FUNCTION_BLOCK SL_Dispense (* Dispense: Requires TRUE; waits Volume / FlowRate s; Invariant TRUE *)
  (* Standard: 61499-2 *)
  (* Version 0.1, 2026-09-28, Project contributors, AAU Smart Production Lab *)
  PACKAGE filling;
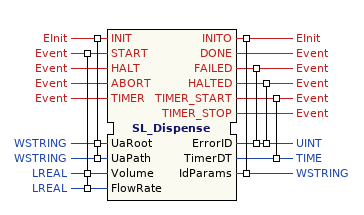
  EVENT_INPUT
    INIT : EInit WITH UaRoot, UaPath;
    START WITH Volume, FlowRate;
    HALT;
    ABORT;
    TIMER;
  END_EVENT
  EVENT_OUTPUT
    INITO : EInit WITH IdParams;
    DONE;
    FAILED WITH ErrorID;
    HALTED WITH ErrorID;
    TIMER_START WITH TimerDT;
    TIMER_STOP;
  END_EVENT
  VAR_INPUT
    UaRoot : WSTRING;
    UaPath : WSTRING;
    Volume : LREAL;
    FlowRate : LREAL;
  END_VAR
  VAR_OUTPUT
    ErrorID : UINT;
    TimerDT : TIME;
    IdParams : WSTRING;
  END_VAR
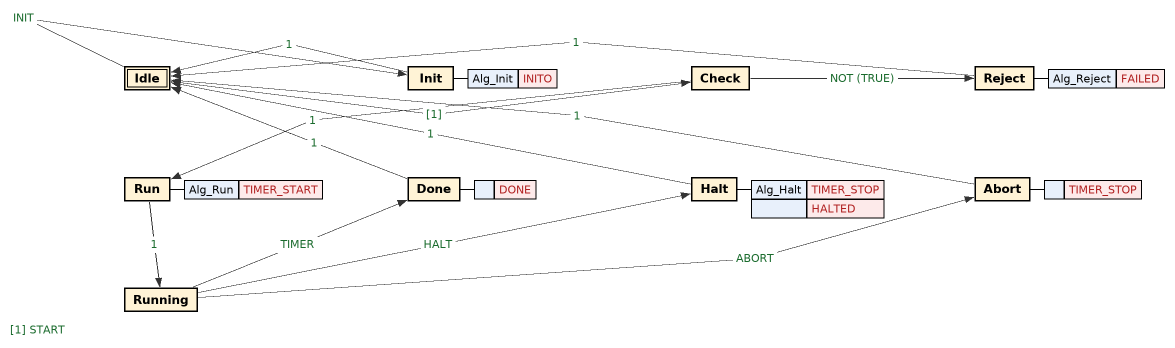
  EC_STATES
    Idle;
    Init : Alg_Init -> INITO;
    Check;
    Reject : Alg_Reject -> FAILED;
    Run : Alg_Run -> TIMER_START;
    Done : -> DONE;
    Halt : Alg_Halt -> TIMER_STOP, -> HALTED;
    Abort : -> TIMER_STOP;
    Running;
  END_STATES
  EC_TRANSITIONS
    Idle TO Init := INIT;
    Init TO Idle := 1;
    Idle TO Check := START;
    Check TO Reject := NOT (TRUE);
    Running TO Done := TIMER;
    Done TO Idle := 1;
    Halt TO Idle := 1;
    Abort TO Idle := 1;
    Check TO Run := 1;
    Run TO Running := 1;
    Running TO Halt := HALT;
    Running TO Abort := ABORT;
    Reject TO Idle := 1;
  END_TRANSITIONS
  ALGORITHM Alg_Init IN ST:
IdParams := CONCAT(CONCAT(CONCAT(CONCAT(CONCAT("opc_ua[WRITE;", CONCAT(UaRoot, UaPath)), "/Parameters/Volume;"), CONCAT(UaRoot, UaPath)), "/Parameters/FlowRate"), "]");
  END_ALGORITHM
  ALGORITHM Alg_Reject IN ST:
ErrorID := 1;
  END_ALGORITHM
  ALGORITHM Alg_Run IN ST:
TimerDT := MUL_TIME(T#1s, Volume / FlowRate);
  END_ALGORITHM
  ALGORITHM Alg_Halt IN ST:
ErrorID := 7;
  END_ALGORITHM
END_FUNCTION_BLOCK
